(* IEC 61131-3 sources: volt/packages/volt-lsp-iec/test-corpus/awa-palletizer/Device/Plc Logic/Application/Library Manager/CmpSettings, 10 files *)

(* ---- SETTGCACHEOPTIONS.gvl ---- *)
VAR_GLOBAL
	CMPSETTINGS_CACHED : DINT := 0;
	CMPSETTINGS_NOT_CACHED : DINT := 1;
END_VAR

(* ---- SETTGBEGINUPDATE.pou ---- *)
FUNCTION SETTGBEGINUPDATE : RTS_IEC_RESULT
END_FUNCTION

(* ---- SETTGENDUPDATE.pou ---- *)
FUNCTION SETTGENDUPDATE : RTS_IEC_RESULT
END_FUNCTION

(* ---- SETTGGETINTVALUE.pou ---- *)
FUNCTION SETTGGETINTVALUE : RTS_IEC_RESULT
VAR_INPUT
	PSZCOMPONENT : REFERENCE TO STRING;
	PSZKEY : REFERENCE TO STRING;
	PIVALUE : POINTER TO DINT;
	IDEFAULT : DINT;
	BCACHED : DINT;
END_VAR
END_FUNCTION

(* ---- SETTGGETSTRINGVALUE.pou ---- *)
FUNCTION SETTGGETSTRINGVALUE : RTS_IEC_RESULT
VAR_INPUT
	PSZCOMPONENT : REFERENCE TO STRING;
	PSZKEY : REFERENCE TO STRING;
	PSZVALUE : POINTER TO STRING;
	PILEN : POINTER TO DINT;
	PSZDEFAULT : REFERENCE TO STRING;
	BCACHED : DINT;
END_VAR
END_FUNCTION

(* ---- SETTGGETWSTRINGVALUE.pou ---- *)
FUNCTION SETTGGETWSTRINGVALUE : RTS_IEC_RESULT
VAR_INPUT
	PSZCOMPONENT : REFERENCE TO STRING;
	PSZKEY : REFERENCE TO STRING;
	PWSZVALUE : POINTER TO WSTRING;
	PILEN : POINTER TO DINT;
	PWSZDEFAULT : REFERENCE TO WSTRING;
	BCACHED : DINT;
END_VAR
END_FUNCTION

(* ---- SETTGREMOVEKEY.pou ---- *)
FUNCTION SETTGREMOVEKEY : RTS_IEC_RESULT
VAR_INPUT
	PSZCOMPONENT : REFERENCE TO STRING;
	PSZKEY : REFERENCE TO STRING;
END_VAR
END_FUNCTION

(* ---- SETTGSETINTVALUE.pou ---- *)
FUNCTION SETTGSETINTVALUE : RTS_IEC_RESULT
VAR_INPUT
	PSZCOMPONENT : REFERENCE TO STRING;
	PSZKEY : REFERENCE TO STRING;
	IVALUE : DINT;
	IBASE : DINT := 10;
END_VAR
END_FUNCTION

(* ---- SETTGSETSTRINGVALUE.pou ---- *)
FUNCTION SETTGSETSTRINGVALUE : RTS_IEC_RESULT
VAR_INPUT
	PSZCOMPONENT : REFERENCE TO STRING;
	PSZKEY : REFERENCE TO STRING;
	PSZVALUE : REFERENCE TO STRING;
	ILEN : DINT;
END_VAR
END_FUNCTION

(* ---- SETTGSETWSTRINGVALUE.pou ---- *)
FUNCTION SETTGSETWSTRINGVALUE : UDINT
VAR_INPUT
	PSZCOMPONENT : REFERENCE TO STRING;
	PSZKEY : REFERENCE TO STRING;
	PWSZVALUE : REFERENCE TO WSTRING;
	ILEN : DINT;
END_VAR
END_FUNCTION
